// TIA Portal V20 export
TYPE "typeUnitCommunicationControlNode"
// stored: Namespace Unit1.Em0
   STRUCT
      BA030 : "Unit1.Em0.typeUnitCommunicationControlNodeBA030";
   END_STRUCT;
END_TYPE
